FUNCTION_BLOCK E_DEMUX_8 (* Event demultiplexer (generic FB) *)
  (* Standard: 61499-1 Annex A; Description: Copyright (c) 2017, 2024 fortiss GmbH, HR Agrartechnik GmbH This program and the accompanying materials are made available under the terms of the Eclipse Public License 2.0 which is available at https://www.eclipse.org/legal/epl-2.0/ SPDX-License-Identifier: EPL-2.0 *)
  (* Version 3.0, 2025-04-14, Patrick Aigner, changed package *)
  (* Version 1.0, 2024-07-15, Franz H??pfinger, HR Agrartechnik GmbH, copy from E_DEMUX and make a E_DEMUX8 in the same way *)
  PACKAGE iec61499::events;
  {SET_ATTRIBUTE(eclipse4diac::core::GenericClassName, 'GEN_E_DEMUX')}
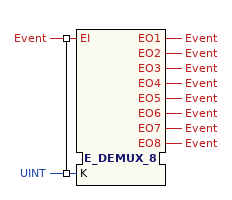
  EVENT_INPUT
    EI WITH K; (* Event to demultiplex *)
  END_EVENT
  EVENT_OUTPUT
    EO1; (* Output, demultiplexed from EI when K=0 *)
    EO2; (* Output, demultiplexed from EI when K=1 *)
    EO3; (* Output, demultiplexed from EI when K=2 *)
    EO4; (* Output, demultiplexed from EI when K=3 *)
    EO5; (* Output, demultiplexed from EI when K=4 *)
    EO6; (* Output, demultiplexed from EI when K=5 *)
    EO7; (* Output, demultiplexed from EI when K=6 *)
    EO8; (* Output, demultiplexed from EI when K=7 *)
  END_EVENT
  VAR_INPUT
    K : UINT; (* Event index *)
  END_VAR
END_FUNCTION_BLOCK
